INTERFACE I_ServerResponse

METHOD PUBLIC Accepted
VAR_INPUT
END_VAR
END_METHOD

METHOD PUBLIC Busy
VAR_INPUT
END_VAR
END_METHOD

METHOD PUBLIC Error
VAR_INPUT
	ErrorCode : T_MAXSTRING;
	Message : T_MAXSTRING;
END_VAR
END_METHOD

PROPERTY PUBLIC Header : I_Header
GET
END_GET
END_PROPERTY

PROPERTY PUBLIC HeadersSent : BOOL
GET
END_GET
END_PROPERTY

METHOD PUBLIC Pending
VAR_INPUT
	ResponseId : REFERENCE TO T_MAXSTRING;
	RetryDelayInMs : UDINT;
END_VAR
END_METHOD

METHOD PUBLIC Success
VAR_INPUT
END_VAR
END_METHOD

METHOD PUBLIC SuccessWithPayload
VAR_INPUT
	PayloadDataAddress : PVOID;
	
	// Number of payload bytes to copy.
    // Does not include the STRING null terminator.
	PayloadDataSize : UDINT;
END_VAR
END_METHOD

END_INTERFACE

(* stored: Version 1.1.0.1, ProductVersion 3.1.4026.18
   Itf I_ServerResponse: Id {73400505-8067-4057-a9de-9d0c6e7226c5}
   Method Accepted: Id {6246fac0-fc8d-4feb-9371-c0177960159c}
   Method Busy: Id {b25a9655-c66e-49ae-baa3-1edf29ea3497}
   Method Error: Id {d237216f-7967-40d2-9412-b4a24b85b267}
   Property Header: Id {8ffc523a-6ad8-4515-8678-65029bb01dfe}
   Get Get: Id {fe96836b-a607-43f6-b9c8-6c3cd3277023}
   Property HeadersSent: Id {69151604-9c1b-4504-8acc-666dace45603}
   Get Get: Id {77ce1403-f79b-43fa-add7-726ec1bd603b}
   Method Pending: Id {020c4672-a442-48d5-8a39-1dc52a2129db}
   Method Success: Id {cdab33a1-e5db-491f-a118-2f8d58ebf253}
   Method SuccessWithPayload: Id {d047699e-ce48-49a9-a850-a788b6066cc8} *)
